// TIA Portal V17 export
// export: Created 2025-03-13T10:31:20.8901656Z, ExportSetting WithDefaults, DisplayName Totally Integrated Automation Portal, DisplayVersion V17 Update 8, DisplayName TIA Portal Openness, DisplayVersion V17 Update 8, DisplayName TIA Portal Version Control Interface, DisplayVersion V17, DisplayName SINAMICS Startdrive Advanced, DisplayVersion V17 SP2, DisplayName SINAMICS Startdrive G110M, G120, G120C, G120D, G120P, G115D, DisplayVersion V17 SP2, DisplayName SINAMICS Startdrive G130, G150, S120, S150, SINAMICS MV, S210, DisplayVersion V17 SP2, DisplayName STEP 7 Professional, DisplayVersion V17 Update 8, DisplayName SINUMERIK ONE STEP 7 Toolbox, DisplayVersion V17 Update 12, DisplayName SINUMERIK 840D sl STEP 7 Toolbox, DisplayVersion V17 Update 12, DisplayName STEP 7 Safety, DisplayVersion V17 Update 6, DisplayName WinCC Advanced, DisplayVersion V17 Update 8
TYPE "MACHINE ALARM"
// stored: IsFailsafeCompliant false
   STRUCT
      IS_ALARMS : Bool;   // IMMEDIATE STOP ALARMS
      RHP_ALARMS : Bool;   // RETURN HOME POSITION ALARMS
      SEOC_ALARMS : Bool;   // STOP END OF CYCLE ALARMS
      IS_WARNING : Bool;   // IMMEDIATE STOP WARNING / IMMEDIATE STOP WARNINGS
      RHP_WARNING : Bool;   // RETURN HOME POSITION WARNING / RETURN HOME POSITION WARNINGS
      SEOC_WARNING : Bool;   // STOP END OF CYCLE WARNING / STOP END OF CYCLE WARNINGS
      WARNING : Bool;   // WARNING / WARNINGS
      HELP : Bool;   // HELP
      aux1_2 : Bool;   // aux1_2
      aux1_3 : Bool;   // aux1_3
      aux1_4 : Bool;   // aux1_4
      aux1_5 : Bool;   // aux1_5
      RHP_DONE_PULSE : Bool;   // RETURN HOME POSITION DONE PULSE
      RHP_DONE : Bool;   // RETURN HOME POSITION DONE
      ALARM : Bool;   // FAULT / ALARM
      RESET_ALL_SEQUENCES : Bool;   // RESET ALL SEQUENCES
      RESET_LOCAL_SEQUENCES : Bool;   // RESET LOCAL SEQUENCES
      RESET_STOP_WARNING : Bool;   // RESET STOP WARNING / RESET STOP WARNINGS
      ALARM_DECODING : DInt;   // FAULT DECODING / ALARMS DECODING
      WARNING_DECODING : DInt;   // WARNING DECODING / WARNINGS DECODING
      HELP_DECODING : DInt;   // HELP DECODING
   END_STRUCT;
END_TYPE
